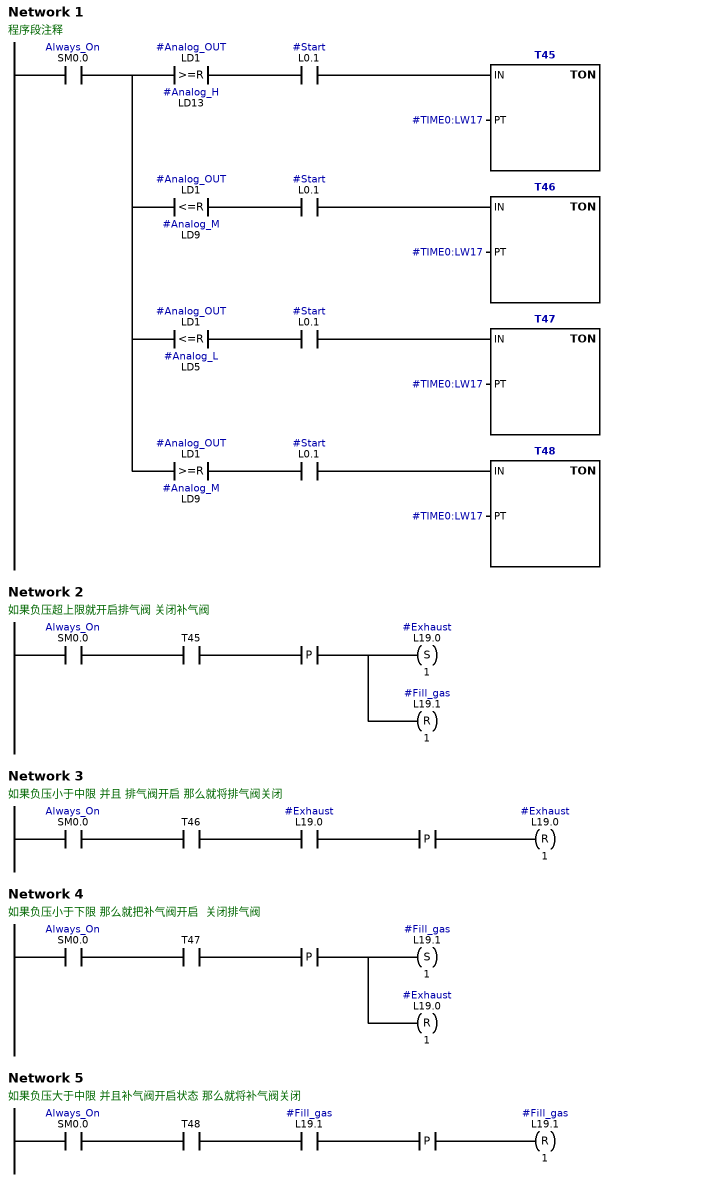
[picture p24: SBR13 networks 1-5]
Network 1
// 程序段注释
LD     Always_On:SM0.0
LPS
AR>=   #Analog_OUT:LD1, #Analog_H:LD13
A      #Start:L0.1
TON    T45, #TIME0:LW17
LRD
AR<=   #Analog_OUT:LD1, #Analog_M:LD9
A      #Start:L0.1
TON    T46, #TIME0:LW17
LRD
AR<=   #Analog_OUT:LD1, #Analog_L:LD5
A      #Start:L0.1
TON    T47, #TIME0:LW17
LPP
AR>=   #Analog_OUT:LD1, #Analog_M:LD9
A      #Start:L0.1
TON    T48, #TIME0:LW17
Network 2
// 如果负压超上限就开启排气阀 关闭补气阀
LD     Always_On:SM0.0
A      T45
EU
S      #Exhaust:L19.0, 1
R      #Fill_gas:L19.1, 1
Network 3
// 如果负压小于中限 并且 排气阀开启 那么就将排气阀关闭
LD     Always_On:SM0.0
A      T46
A      #Exhaust:L19.0
EU
R      #Exhaust:L19.0, 1
Network 4
// 如果负压小于下限 那么就把补气阀开启  关闭排气阀
LD     Always_On:SM0.0
A      T47
EU
S      #Fill_gas:L19.1, 1
R      #Exhaust:L19.0, 1
Network 5
// 如果负压大于中限 并且补气阀开启状态 那么就将补气阀关闭 
LD     Always_On:SM0.0
A      T48
A      #Fill_gas:L19.1
EU
R      #Fill_gas:L19.1, 1
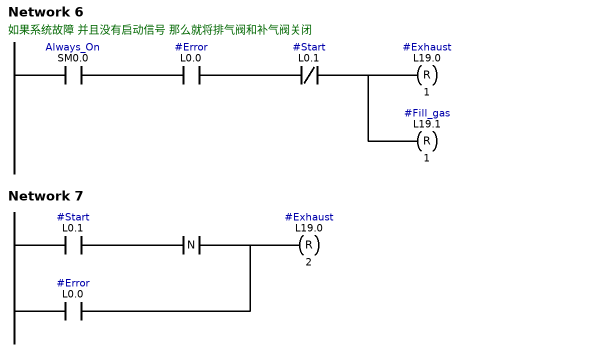
Network 6
// 如果系统故障 并且没有启动信号 那么就将排气阀和补气阀关闭
LD     Always_On:SM0.0
A      #Error:L0.0
AN     #Start:L0.1
R      #Exhaust:L19.0, 1
R      #Fill_gas:L19.1, 1
Network 7
LD     #Start:L0.1
ED
O      #Error:L0.0
R      #Exhaust:L19.0, 2
END_SUBROUTINE_BLOCK

SUBROUTINE_BLOCK 混料程序:SBR14
TITLE=1.	混合机启动程序:做按钮单独启停控制(实现批混模式)
// 
// 2.	混合机进料状态，达到重量大于1000kg（可调）延时ＸＸＳ
// 　　　    进入混合状态，停止输出混合要料信号．
// 
// 3.	混合状态（混合时间可调），显示混料时间，做倒计时。
// 
// 4.	混料完成信号，（运行出料）
// 
// 5.	出料达到设定出料下限下于100ｋｇ（可调）延时XXS，再次进入混料进料状态。
//                 需要显示混料机的状态，（进料，混合计时，出料）
// 
VAR_INPUT
Star:BOOL;	// L0.0 混合机启动
MixmotorWeight:DWORD;	// LD1 混合机重量读取
WeightH:DWORD;	// LD5 混合机重量上限
WeightL:DWORD;	// LD9 混合机重量下限
DelayH:WORD;	// LW13 上限延时
DelayL:WORD;	// LW15 下限延时
MixtimeSet:WORD;	// LW17 混合时间设置
END_VAR
VAR_IN_OUT
FeedState:BOOL;	// L19.0 进料状态
MixState:BOOL;	// L19.1 混合状态
OutState:BOOL;	// L19.2 出料状态
Countdown:WORD;	// LW20 混合倒计时
MixMotor:BOOL;	// L22.0 混合机电机
OutDone:BOOL;	// L22.1 出料完成
END_VAR
BEGIN
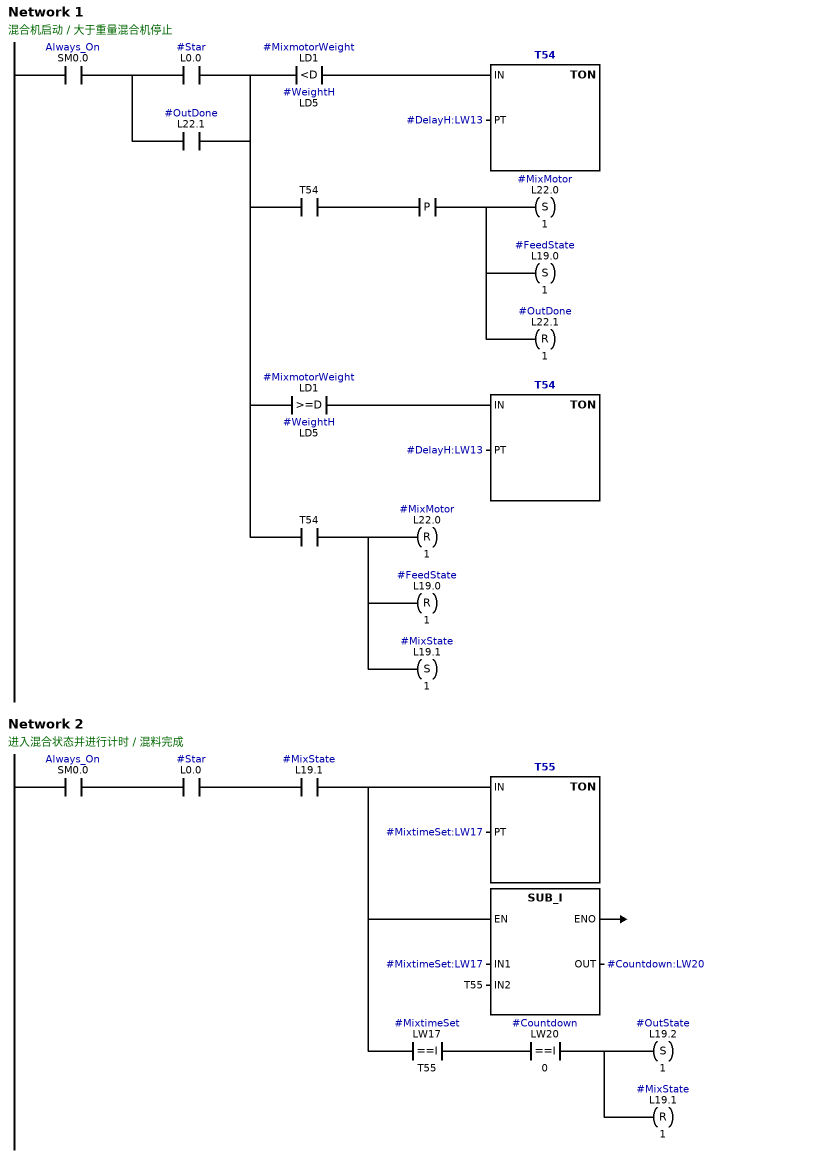
Network 1
// 混合机启动
// 大于重量混合机停止
LD     Always_On:SM0.0
LD     #Star:L0.0
O      #OutDone:L22.1
ALD
LPS
AD<    #MixmotorWeight:LD1, #WeightH:LD5
TON    T54, #DelayH:LW13
LRD
A      T54
EU
S      #MixMotor:L22.0, 1
S      #FeedState:L19.0, 1
R      #OutDone:L22.1, 1
LRD
AD>=   #MixmotorWeight:LD1, #WeightH:LD5
TON    T54, #DelayH:LW13
LPP
A      T54
R      #MixMotor:L22.0, 1
R      #FeedState:L19.0, 1
S      #MixState:L19.1, 1
Network 2
// 进入混合状态并进行计时
// 混料完成
LD     Always_On:SM0.0
A      #Star:L0.0
A      #MixState:L19.1
TON    T55, #MixtimeSet:LW17
MOVW   #MixtimeSet:LW17, #Countdown:LW20
-I     T55, #Countdown:LW20
AW=    #MixtimeSet:LW17, T55
AW=    #Countdown:LW20, 0
S      #OutState:L19.2, 1
R      #MixState:L19.1, 1
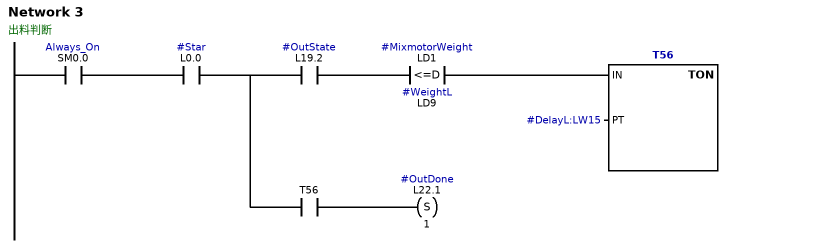
Network 3
// 出料判断
LD     Always_On:SM0.0
A      #Star:L0.0
LPS
A      #OutState:L19.2
AD<=   #MixmotorWeight:LD1, #WeightL:LD9
TON    T56, #DelayL:LW15
LPP
A      T56
S      #OutDone:L22.1, 1
END_SUBROUTINE_BLOCK

SUBROUTINE_BLOCK 系统泄压程序:SBR15
TITLE=
VAR_INPUT
Start:BOOL;	// L0.0 
OUT_Analog:REAL;	// LD1 
END_VAR
VAR_IN_OUT
Date_set_FH:REAL;	// LD5 
Date_set_FL:REAL;	// LD9 
Date_set_ZH:REAL;	// LD13 
Date_set_ZL:REAL;	// LD17 
Auto_OUT:BOOL;	// L21.0 
END_VAR
VAR
Auto_16A:BOOL;	// L21.1 中间变量1
Auto_16B:BOOL;	// L21.2 中间变量2
END_VAR
BEGIN
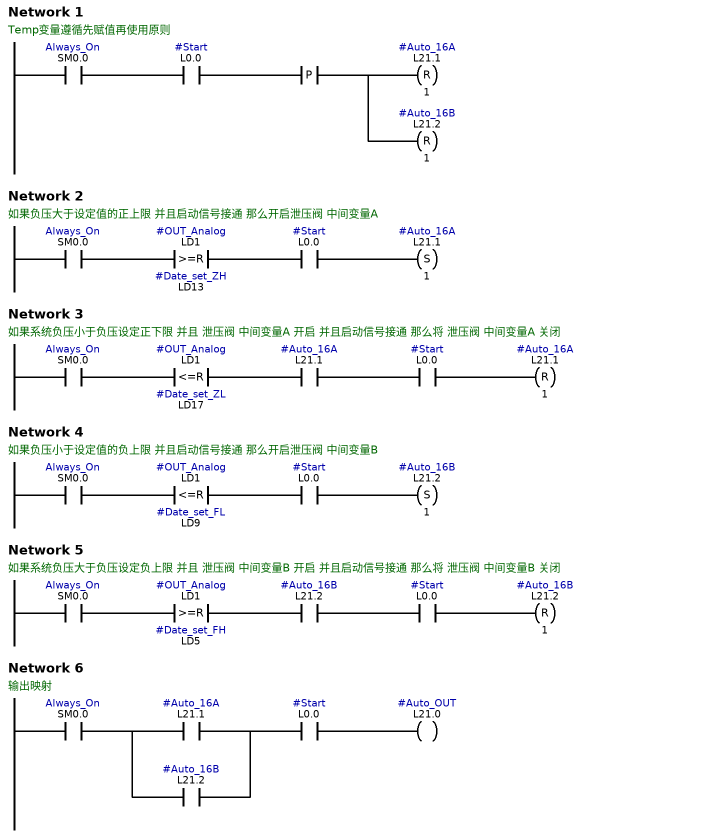
Network 1
// Temp变量遵循先赋值再使用原则
LD     Always_On:SM0.0
A      #Start:L0.0
EU
R      #Auto_16A:L21.1, 1
R      #Auto_16B:L21.2, 1
Network 2
// 如果负压大于设定值的正上限 并且启动信号接通 那么开启泄压阀 中间变量A
LD     Always_On:SM0.0
AR>=   #OUT_Analog:LD1, #Date_set_ZH:LD13
A      #Start:L0.0
S      #Auto_16A:L21.1, 1
Network 3
// 如果系统负压小于负压设定正下限 并且 泄压阀 中间变量A 开启 并且启动信号接通 那么将 泄压阀 中间变量A 关闭
LD     Always_On:SM0.0
AR<=   #OUT_Analog:LD1, #Date_set_ZL:LD17
A      #Auto_16A:L21.1
A      #Start:L0.0
R      #Auto_16A:L21.1, 1
Network 4
// 如果负压小于设定值的负上限 并且启动信号接通 那么开启泄压阀 中间变量B
LD     Always_On:SM0.0
AR<=   #OUT_Analog:LD1, #Date_set_FL:LD9
A      #Start:L0.0
S      #Auto_16B:L21.2, 1
Network 5
// 如果系统负压大于负压设定负上限 并且 泄压阀 中间变量B 开启 并且启动信号接通 那么将 泄压阀 中间变量B 关闭
LD     Always_On:SM0.0
AR>=   #OUT_Analog:LD1, #Date_set_FH:LD5
A      #Auto_16B:L21.2
A      #Start:L0.0
R      #Auto_16B:L21.2, 1
Network 6
// 输出映射
LD     Always_On:SM0.0
LD     #Auto_16A:L21.1
O      #Auto_16B:L21.2
ALD
A      #Start:L0.0
=      #Auto_OUT:L21.0
END_SUBROUTINE_BLOCK

SUBROUTINE_BLOCK 仓泵1:SBR16
TITLE=
VAR_INPUT
IN_LW:BOOL;	// L0.0 上料位信号
END_VAR
VAR_IN_OUT
呼吸阀:BOOL;	// L0.1 
进料阀:BOOL;	// L0.2 
进料阀上:BOOL;	// L0.3 
仓顶阀:BOOL;	// L0.4 
硫化阀:BOOL;	// L0.5 
输送阀:BOOL;	// L0.6 
疏通阀:BOOL;	// L0.7 
出口阀:BOOL;	// L1.0 
切换阀:BOOL;	// L1.1 
END_VAR
BEGIN
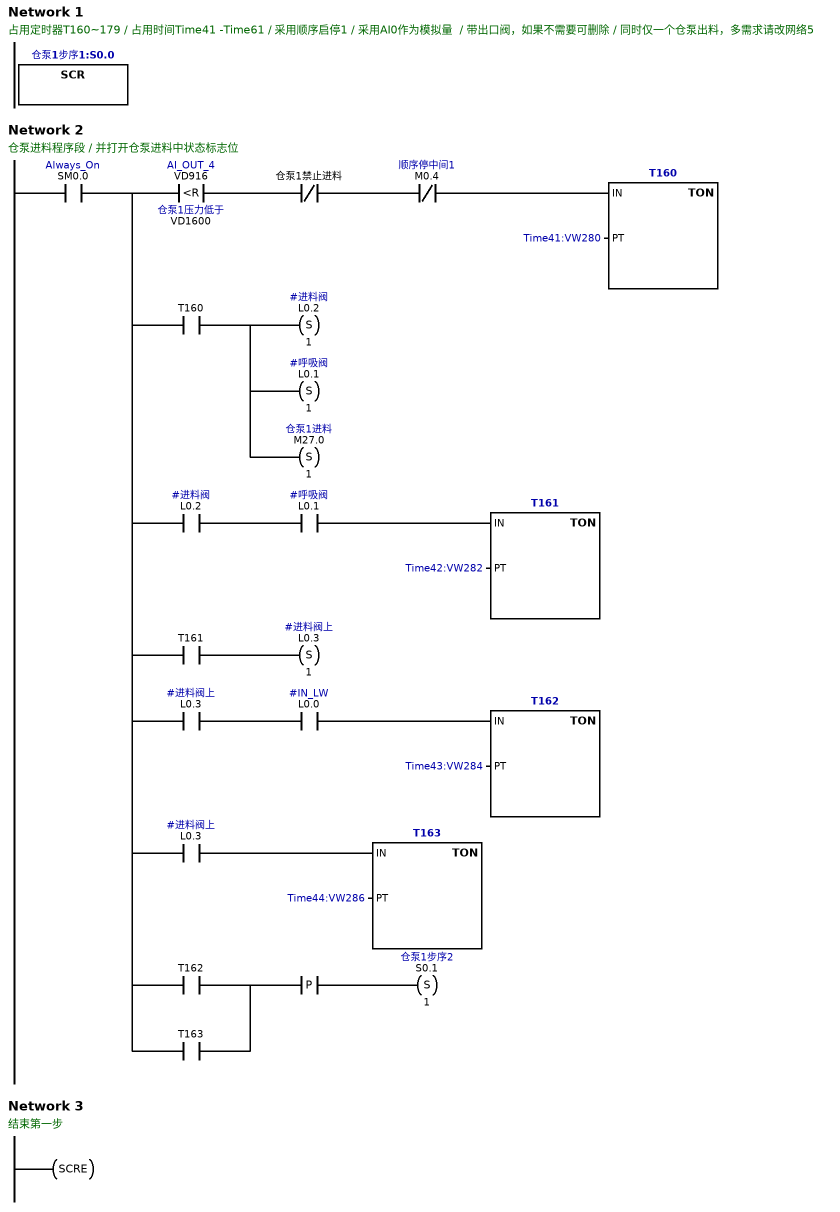
Network 1
// 占用定时器T160~179
// 占用时间Time41 -Time61
// 采用顺序启停1
// 采用AI0作为模拟量 
// 带出口阀，如果不需要可删除
// 同时仅一个仓泵出料，多需求请改网络5
LSCR   仓泵1步序1:S0.0
Network 2
// 仓泵进料程序段
// 并打开仓泵进料中状态标志位
// (network saved uncompiled; LAD cells follow)
// row 0: c0 -| |- Always_On:SM0.0 v  c1 -|<R|- AI_OUT_4:VD916, 仓泵1压力低于:VD1600  c2 -|/|- 仓泵1禁止进料  c3 -|/|- 顺序停中间1:M0.4  c4 --  c5 [TON T160 IN:=power@row0, PT:=Time41:VW280]
// row 1: c0 ^v  c5 [box]
// row 2: c0 ^v  c1 -| |- T160 v  c2 -(S) #进料阀:L0.2, 1
// row 3: c0 ^v  c1 ^v  c2 -(S) #呼吸阀:L0.1, 1
// row 4: c0 ^v  c1 ^  c2 -(S) 仓泵1进料:M27.0, 1
// row 5: c0 ^v  c1 -| |- #进料阀:L0.2  c2 -| |- #呼吸阀:L0.1  c3 --  c4 [TON T161 IN:=power@row5, PT:=Time42:VW282]
// row 6: c0 ^v  c4 [box]
// row 7: c0 ^v  c1 -| |- T161  c2 -(S) #进料阀上:L0.3, 1
// row 8: c0 ^v  c1 -| |- #进料阀上:L0.3  c2 -| |- #IN_LW:L0.0  c3 --  c4 [TON T162 IN:=power@row8, PT:=Time43:VW284]
// row 9: c0 ^v  c4 [box]
// row 10: c0 ^v  c1 -| |- #进料阀上:L0.3  c2 --  c3 [TON T163 IN:=power@row10, PT:=Time44:VW286]
// row 11: c0 ^v  c3 [box]
// row 12: c0 ^v  c1 -| |- T162 v  c2 -|P|-  c3 -(S) 仓泵1步序2:S0.1, 1
// row 13: c0 ^  c1 -| |- T163 ^
Network 3
// 结束第一步
SCRE
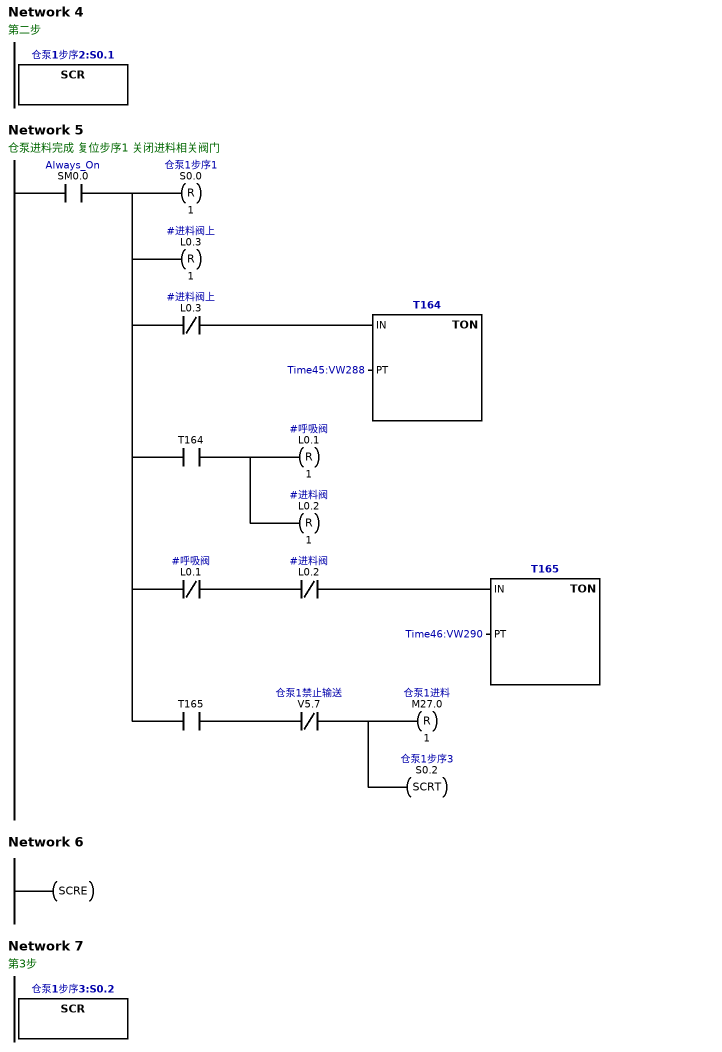
Network 4
// 第二步 
LSCR   仓泵1步序2:S0.1
Network 5
// 仓泵进料完成 复位步序1 关闭进料相关阀门
LD     Always_On:SM0.0
LPS
R      仓泵1步序1:S0.0, 1
R      #进料阀上:L0.3, 1
AN     #进料阀上:L0.3
TON    T164, Time45:VW288
LRD
A      T164
R      #呼吸阀:L0.1, 1
R      #进料阀:L0.2, 1
LRD
AN     #呼吸阀:L0.1
AN     #进料阀:L0.2
TON    T165, Time46:VW290
LPP
A      T165
AN     仓泵1禁止输送:V5.7
R      仓泵1进料:M27.0, 1
SCRT   仓泵1步序3:S0.2
Network 6
SCRE
Network 7
// 第3步 
LSCR   仓泵1步序3:S0.2
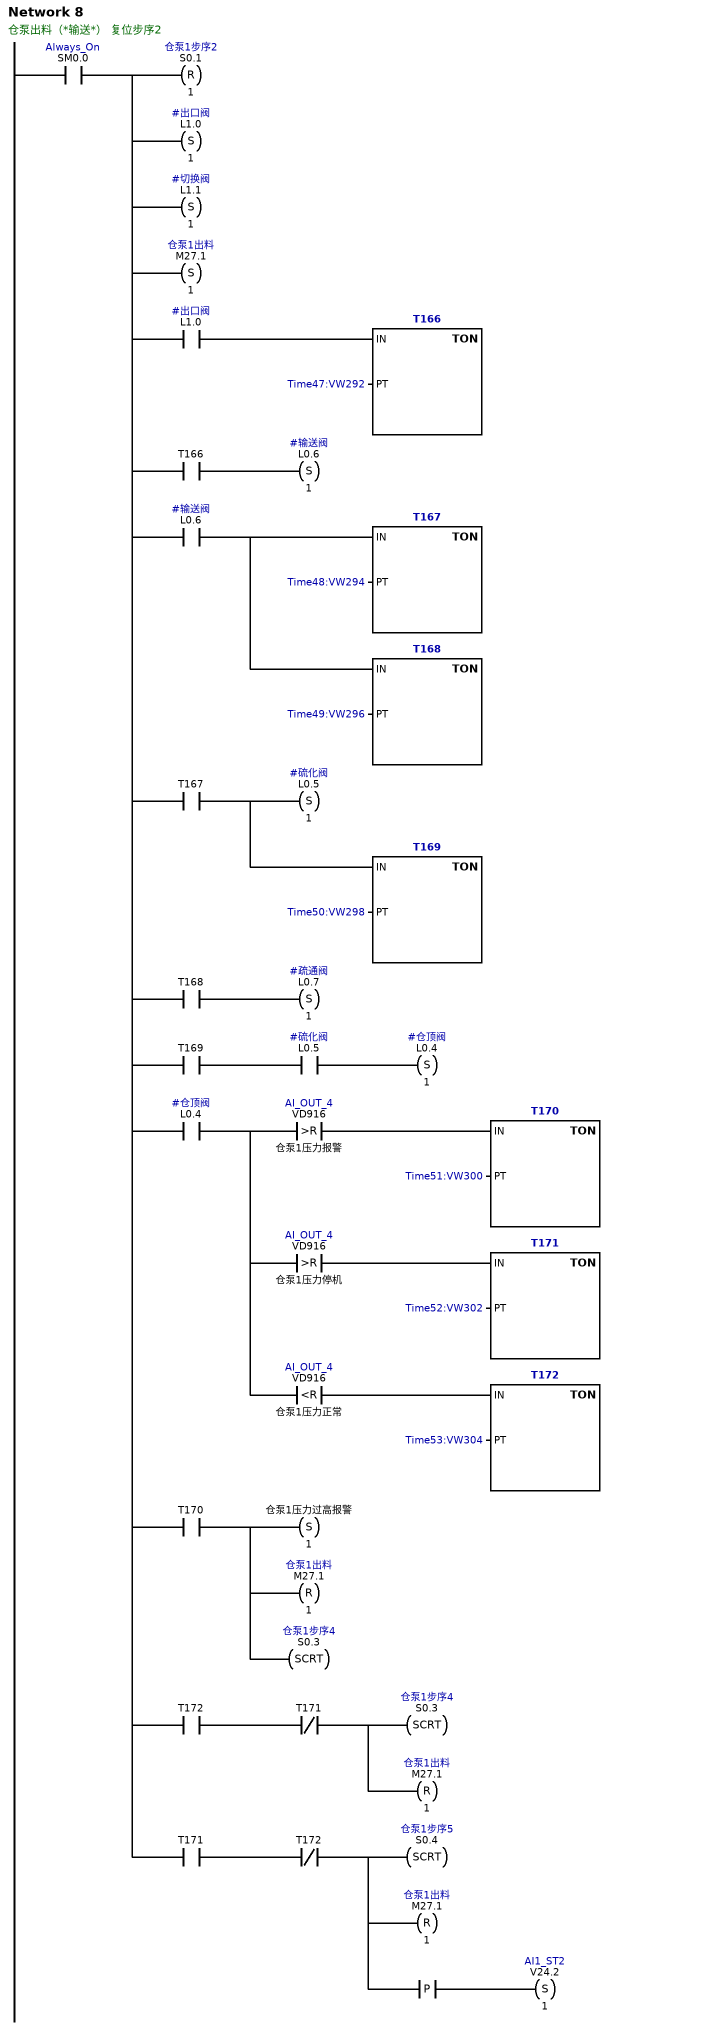
Network 8
// 仓泵出料（*输送*） 复位步序2
// (network saved uncompiled; LAD cells follow)
// row 0: c0 -| |- Always_On:SM0.0 v  c1 -(R) 仓泵1步序2:S0.1, 1
// row 1: c0 ^v  c1 -(S) #出口阀:L1.0, 1
// row 2: c0 ^v  c1 -(S) #切换阀:L1.1, 1
// row 3: c0 ^v  c1 -(S) 仓泵1出料:M27.1, 1
// row 4: c0 ^v  c1 -| |- #出口阀:L1.0  c2 --  c3 [TON T166 IN:=power@row4, PT:=Time47:VW292]
// row 5: c0 ^v  c3 [box]
// row 6: c0 ^v  c1 -| |- T166  c2 -(S) #输送阀:L0.6, 1
// row 7: c0 ^v  c1 -| |- #输送阀:L0.6 v  c2 --  c3 [TON T167 IN:=power@row7, PT:=Time48:VW294]
// row 8: c0 ^v  c1 ^v  c3 [box]
// row 9: c0 ^v  c1 ^  c2 --  c3 [TON T168 IN:=power@row9, PT:=Time49:VW296]
// row 10: c0 ^v  c3 [box]
// row 11: c0 ^v  c1 -| |- T167 v  c2 -(S) #硫化阀:L0.5, 1
// row 12: c0 ^v  c1 ^  c2 --  c3 [TON T169 IN:=power@row12, PT:=Time50:VW298]
// row 13: c0 ^v  c3 [box]
// row 14: c0 ^v  c1 -| |- T168  c2 -(S) #疏通阀:L0.7, 1
// row 15: c0 ^v  c1 -| |- T169  c2 -| |- #硫化阀:L0.5  c3 -(S) #仓顶阀:L0.4, 1
// row 16: c0 ^v  c1 -| |- #仓顶阀:L0.4 v  c2 -|>R|- AI_OUT_4:VD916, 仓泵1压力报警  c3 --  c4 [TON T170 IN:=power@row16, PT:=Time51:VW300]
// row 17: c0 ^v  c1 ^v  c4 [box]
// row 18: c0 ^v  c1 ^v  c2 -|>R|- AI_OUT_4:VD916, 仓泵1压力停机  c3 --  c4 [TON T171 IN:=power@row18, PT:=Time52:VW302]
// row 19: c0 ^v  c1 ^v  c4 [box]
// row 20: c0 ^v  c1 ^  c2 -|<R|- AI_OUT_4:VD916, 仓泵1压力正常  c3 --  c4 [TON T172 IN:=power@row20, PT:=Time53:VW304]
// row 21: c0 ^v  c4 [box]
// row 22: c0 ^v  c1 -| |- T170 v  c2 -(S) 仓泵1压力过高报警, 1
// row 23: c0 ^v  c1 ^v  c2 -(R) 仓泵1出料:M27.1, 1
// row 24: c0 ^v  c1 ^  c2 -(SCRT) 仓泵1步序4:S0.3
// row 25: c0 ^v  c1 -| |- T172  c2 -|/|- T171 v  c3 -(SCRT) 仓泵1步序4:S0.3
// row 26: c0 ^v  c2 ^  c3 -(R) 仓泵1出料:M27.1, 1
// row 27: c0 ^  c1 -| |- T171  c2 -|/|- T172 v  c3 -(SCRT) 仓泵1步序5:S0.4
// row 28: c2 ^v  c3 -(R) 仓泵1出料:M27.1, 1
// row 29: c2 ^  c3 -|P|-  c4 -(S) AI1_ST2:V24.2, 1
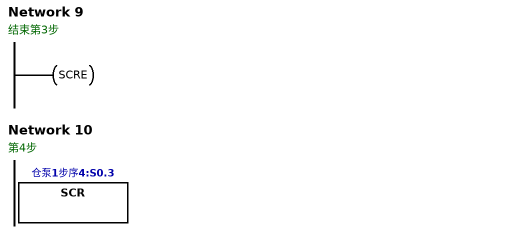
Network 9
// 结束第3步
SCRE
Network 10
// 第4步 
LSCR   仓泵1步序4:S0.3
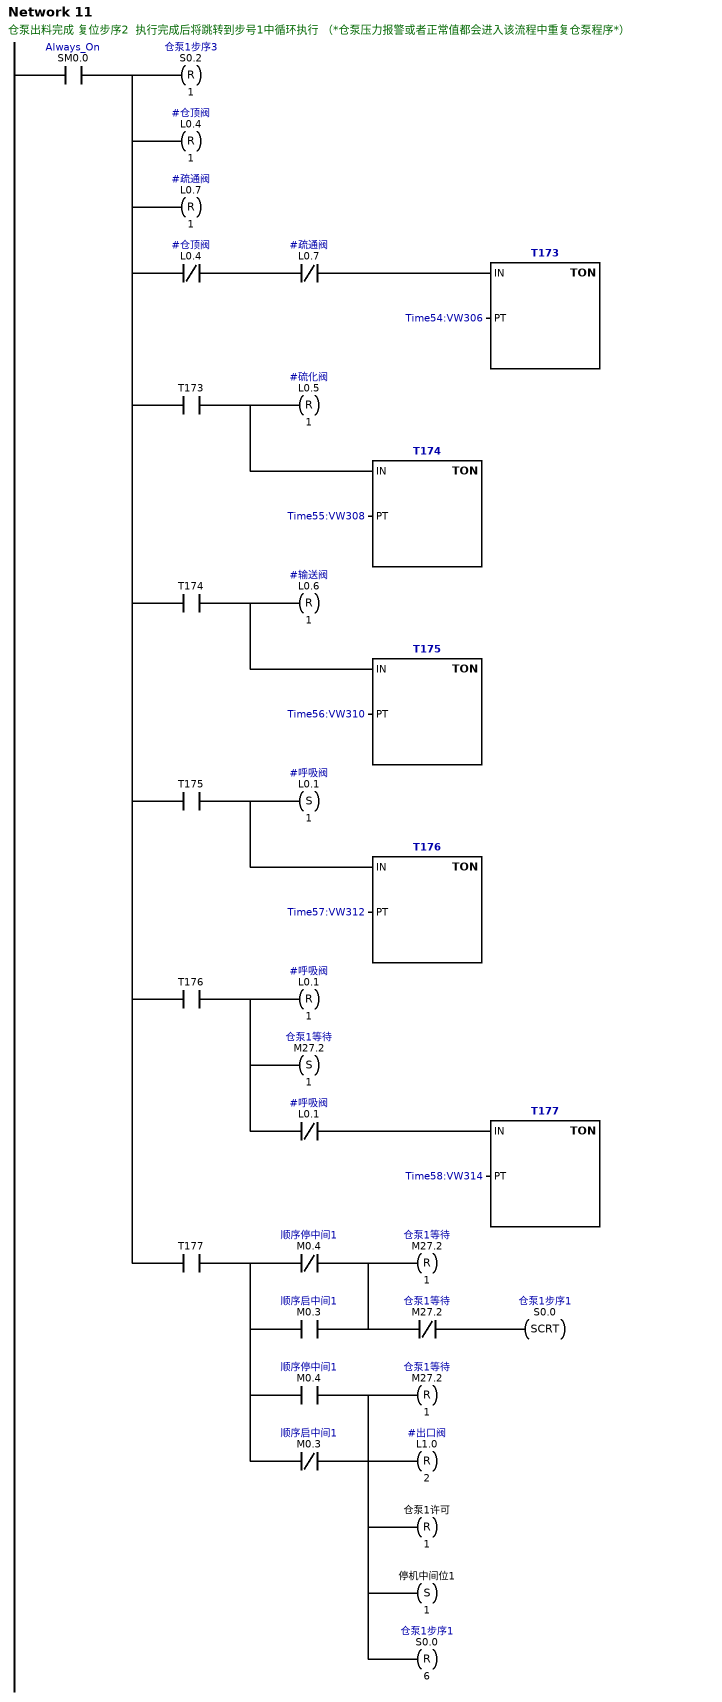
Network 11
// 仓泵出料完成 复位步序2  执行完成后将跳转到步号1中循环执行 （*仓泵压力报警或者正常值都会进入该流程中重复仓泵程序*）
// (network saved uncompiled; LAD cells follow)
// row 0: c0 -| |- Always_On:SM0.0 v  c1 -(R) 仓泵1步序3:S0.2, 1
// row 1: c0 ^v  c1 -(R) #仓顶阀:L0.4, 1
// row 2: c0 ^v  c1 -(R) #疏通阀:L0.7, 1
// row 3: c0 ^v  c1 -|/|- #仓顶阀:L0.4  c2 -|/|- #疏通阀:L0.7  c3 --  c4 [TON T173 IN:=power@row3, PT:=Time54:VW306]
// row 4: c0 ^v  c4 [box]
// row 5: c0 ^v  c1 -| |- T173 v  c2 -(R) #硫化阀:L0.5, 1
// row 6: c0 ^v  c1 ^  c2 --  c3 [TON T174 IN:=power@row6, PT:=Time55:VW308]
// row 7: c0 ^v  c3 [box]
// row 8: c0 ^v  c1 -| |- T174 v  c2 -(R) #输送阀:L0.6, 1
// row 9: c0 ^v  c1 ^  c2 --  c3 [TON T175 IN:=power@row9, PT:=Time56:VW310]
// row 10: c0 ^v  c3 [box]
// row 11: c0 ^v  c1 -| |- T175 v  c2 -(S) #呼吸阀:L0.1, 1
// row 12: c0 ^v  c1 ^  c2 --  c3 [TON T176 IN:=power@row12, PT:=Time57:VW312]
// row 13: c0 ^v  c3 [box]
// row 14: c0 ^v  c1 -| |- T176 v  c2 -(R) #呼吸阀:L0.1, 1
// row 15: c0 ^v  c1 ^v  c2 -(S) 仓泵1等待:M27.2, 1
// row 16: c0 ^v  c1 ^  c2 -|/|- #呼吸阀:L0.1  c3 --  c4 [TON T177 IN:=power@row16, PT:=Time58:VW314]
// row 17: c0 ^v  c4 [box]
// row 18: c0 ^  c1 -| |- T177 v  c2 -|/|- 顺序停中间1:M0.4 v  c3 -(R) 仓泵1等待:M27.2, 1
// row 19: c1 ^v  c2 -| |- 顺序启中间1:M0.3 ^  c3 -|/|- 仓泵1等待:M27.2  c4 -(SCRT) 仓泵1步序1:S0.0
// row 20: c1 ^v  c2 -| |- 顺序停中间1:M0.4 v  c3 -(R) 仓泵1等待:M27.2, 1
// row 21: c1 ^  c2 -|/|- 顺序启中间1:M0.3 ^v  c3 -(R) #出口阀:L1.0, 2
// row 22: c2 ^v  c3 -(R) 仓泵1许可, 1
// row 23: c2 ^v  c3 -(S) 停机中间位1, 1
// row 24: c2 ^  c3 -(R) 仓泵1步序1:S0.0, 6
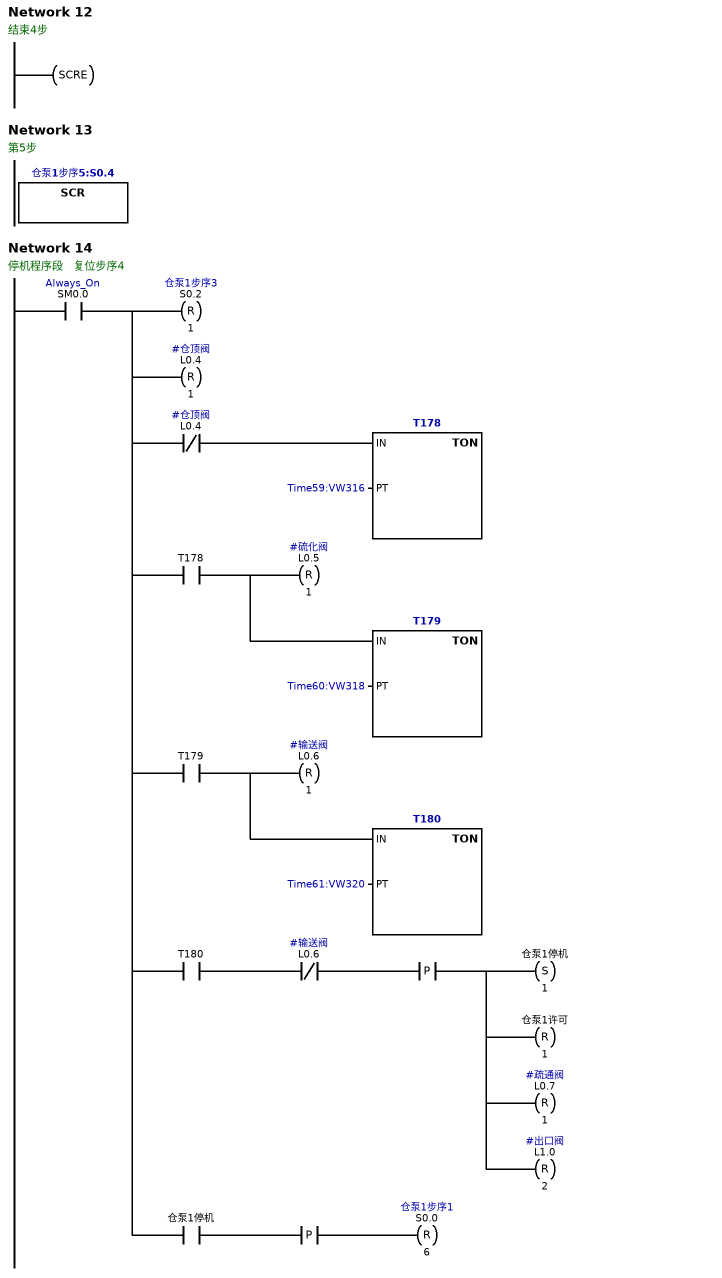
Network 12
// 结束4步
SCRE
Network 13
// 第5步 
LSCR   仓泵1步序5:S0.4
Network 14
// 停机程序段   复位步序4 
// (network saved uncompiled; LAD cells follow)
// row 0: c0 -| |- Always_On:SM0.0 v  c1 -(R) 仓泵1步序3:S0.2, 1
// row 1: c0 ^v  c1 -(R) #仓顶阀:L0.4, 1
// row 2: c0 ^v  c1 -|/|- #仓顶阀:L0.4  c2 --  c3 [TON T178 IN:=power@row2, PT:=Time59:VW316]
// row 3: c0 ^v  c3 [box]
// row 4: c0 ^v  c1 -| |- T178 v  c2 -(R) #硫化阀:L0.5, 1
// row 5: c0 ^v  c1 ^  c2 --  c3 [TON T179 IN:=power@row5, PT:=Time60:VW318]
// row 6: c0 ^v  c3 [box]
// row 7: c0 ^v  c1 -| |- T179 v  c2 -(R) #输送阀:L0.6, 1
// row 8: c0 ^v  c1 ^  c2 --  c3 [TON T180 IN:=power@row8, PT:=Time61:VW320]
// row 9: c0 ^v  c3 [box]
// row 10: c0 ^v  c1 -| |- T180  c2 -|/|- #输送阀:L0.6  c3 -|P|-  v  c4 -(S) 仓泵1停机, 1
// row 11: c0 ^v  c3 ^v  c4 -(R) 仓泵1许可, 1
// row 12: c0 ^v  c3 ^v  c4 -(R) #疏通阀:L0.7, 1
// row 13: c0 ^v  c3 ^  c4 -(R) #出口阀:L1.0, 2
// row 14: c0 ^  c1 -| |- 仓泵1停机  c2 -|P|-  c3 -(R) 仓泵1步序1:S0.0, 6
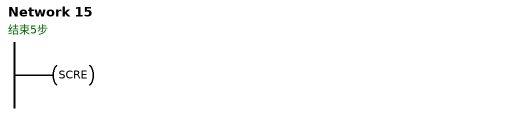
Network 15
// 结束5步
SCRE
END_SUBROUTINE_BLOCK

SUBROUTINE_BLOCK 仓泵2:SBR17
TITLE=
VAR_INPUT
IN_LW:BOOL;	// L0.0 上料位信号
END_VAR
VAR_IN_OUT
呼吸阀:BOOL;	// L0.1 
进料阀:BOOL;	// L0.2 
进料阀上:BOOL;	// L0.3 
仓顶阀:BOOL;	// L0.4 
硫化阀:BOOL;	// L0.5 
输送阀:BOOL;	// L0.6 
疏通阀:BOOL;	// L0.7 
出口阀:BOOL;	// L1.0 
切换阀:BOOL;	// L1.1 
END_VAR
BEGIN
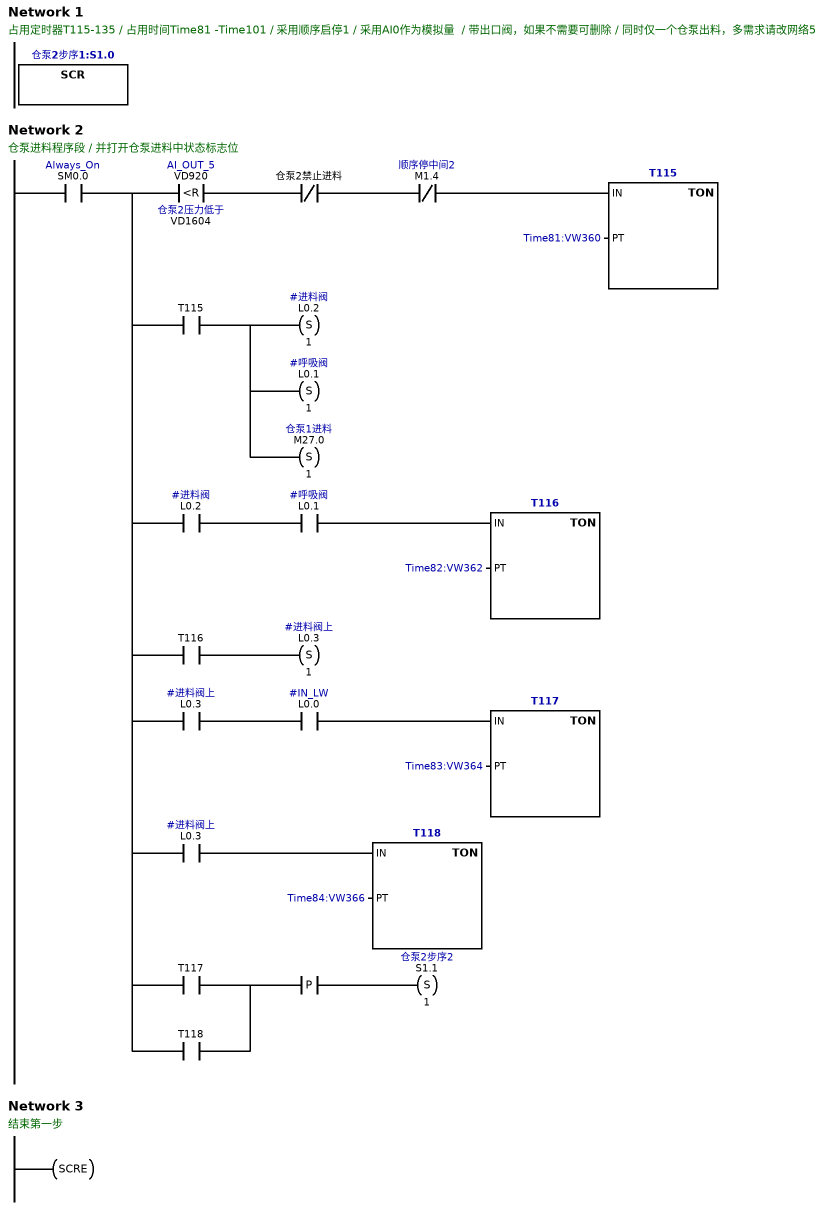
Network 1
// 占用定时器T115-135
// 占用时间Time81 -Time101
// 采用顺序启停1
// 采用AI0作为模拟量 
// 带出口阀，如果不需要可删除
// 同时仅一个仓泵出料，多需求请改网络5
LSCR   仓泵2步序1:S1.0
Network 2
// 仓泵进料程序段
// 并打开仓泵进料中状态标志位
// (network saved uncompiled; LAD cells follow)
// row 0: c0 -| |- Always_On:SM0.0 v  c1 -|<R|- AI_OUT_5:VD920, 仓泵2压力低于:VD1604  c2 -|/|- 仓泵2禁止进料  c3 -|/|- 顺序停中间2:M1.4  c4 --  c5 [TON T115 IN:=power@row0, PT:=Time81:VW360]
// row 1: c0 ^v  c5 [box]
// row 2: c0 ^v  c1 -| |- T115 v  c2 -(S) #进料阀:L0.2, 1
// row 3: c0 ^v  c1 ^v  c2 -(S) #呼吸阀:L0.1, 1
// row 4: c0 ^v  c1 ^  c2 -(S) 仓泵1进料:M27.0, 1
// row 5: c0 ^v  c1 -| |- #进料阀:L0.2  c2 -| |- #呼吸阀:L0.1  c3 --  c4 [TON T116 IN:=power@row5, PT:=Time82:VW362]
// row 6: c0 ^v  c4 [box]
// row 7: c0 ^v  c1 -| |- T116  c2 -(S) #进料阀上:L0.3, 1
// row 8: c0 ^v  c1 -| |- #进料阀上:L0.3  c2 -| |- #IN_LW:L0.0  c3 --  c4 [TON T117 IN:=power@row8, PT:=Time83:VW364]
// row 9: c0 ^v  c4 [box]
// row 10: c0 ^v  c1 -| |- #进料阀上:L0.3  c2 --  c3 [TON T118 IN:=power@row10, PT:=Time84:VW366]
// row 11: c0 ^v  c3 [box]
// row 12: c0 ^v  c1 -| |- T117 v  c2 -|P|-  c3 -(S) 仓泵2步序2:S1.1, 1
// row 13: c0 ^  c1 -| |- T118 ^
Network 3
// 结束第一步
SCRE
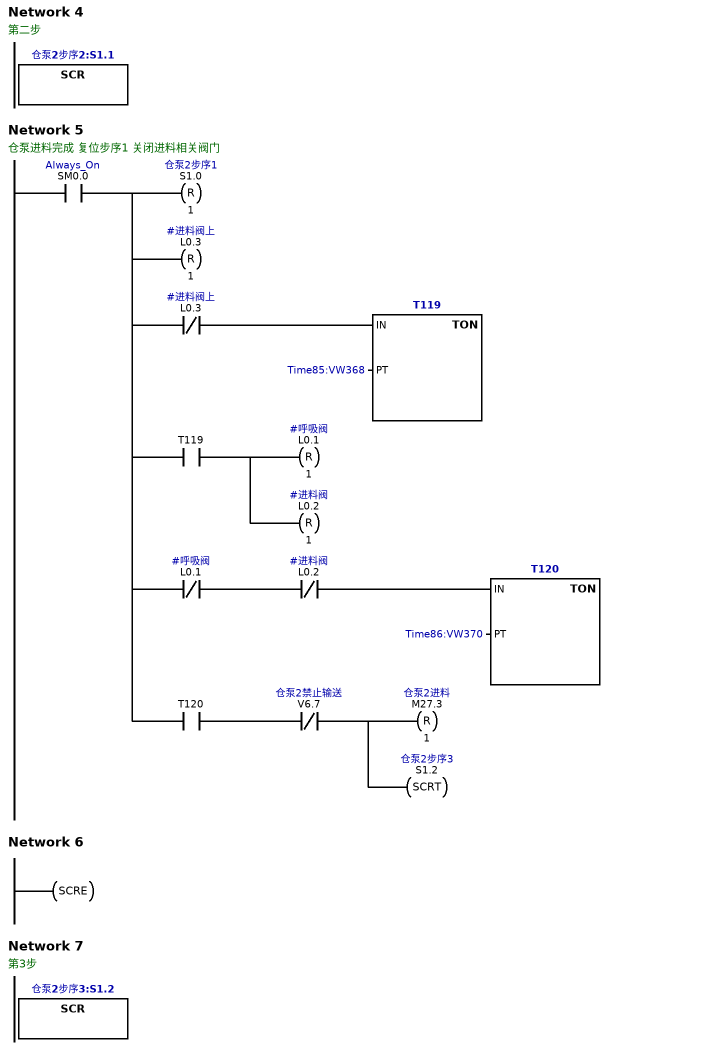
Network 4
// 第二步 
LSCR   仓泵2步序2:S1.1
Network 5
// 仓泵进料完成 复位步序1 关闭进料相关阀门
LD     Always_On:SM0.0
LPS
R      仓泵2步序1:S1.0, 1
R      #进料阀上:L0.3, 1
AN     #进料阀上:L0.3
TON    T119, Time85:VW368
LRD
A      T119
R      #呼吸阀:L0.1, 1
R      #进料阀:L0.2, 1
LRD
AN     #呼吸阀:L0.1
AN     #进料阀:L0.2
TON    T120, Time86:VW370
LPP
A      T120
AN     仓泵2禁止输送:V6.7
R      仓泵2进料:M27.3, 1
SCRT   仓泵2步序3:S1.2
Network 6
SCRE
Network 7
// 第3步 
LSCR   仓泵2步序3:S1.2
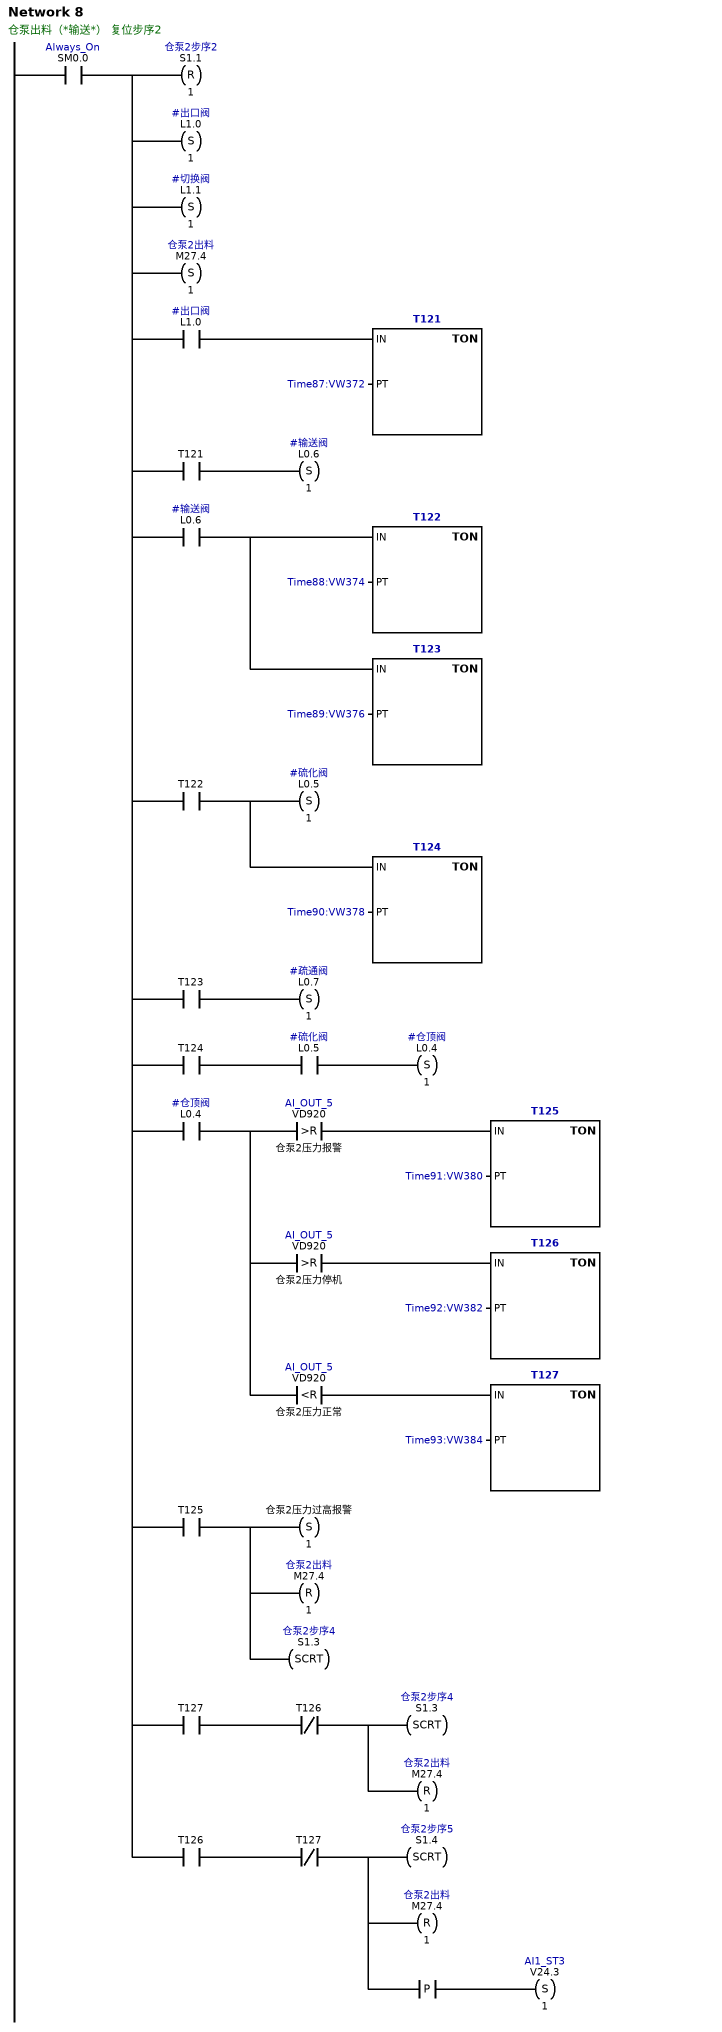
Network 8
// 仓泵出料（*输送*） 复位步序2
// (network saved uncompiled; LAD cells follow)
// row 0: c0 -| |- Always_On:SM0.0 v  c1 -(R) 仓泵2步序2:S1.1, 1
// row 1: c0 ^v  c1 -(S) #出口阀:L1.0, 1
// row 2: c0 ^v  c1 -(S) #切换阀:L1.1, 1
// row 3: c0 ^v  c1 -(S) 仓泵2出料:M27.4, 1
// row 4: c0 ^v  c1 -| |- #出口阀:L1.0  c2 --  c3 [TON T121 IN:=power@row4, PT:=Time87:VW372]
// row 5: c0 ^v  c3 [box]
// row 6: c0 ^v  c1 -| |- T121  c2 -(S) #输送阀:L0.6, 1
// row 7: c0 ^v  c1 -| |- #输送阀:L0.6 v  c2 --  c3 [TON T122 IN:=power@row7, PT:=Time88:VW374]
// row 8: c0 ^v  c1 ^v  c3 [box]
// row 9: c0 ^v  c1 ^  c2 --  c3 [TON T123 IN:=power@row9, PT:=Time89:VW376]
// row 10: c0 ^v  c3 [box]
// row 11: c0 ^v  c1 -| |- T122 v  c2 -(S) #硫化阀:L0.5, 1
// row 12: c0 ^v  c1 ^  c2 --  c3 [TON T124 IN:=power@row12, PT:=Time90:VW378]
// row 13: c0 ^v  c3 [box]
// row 14: c0 ^v  c1 -| |- T123  c2 -(S) #疏通阀:L0.7, 1
// row 15: c0 ^v  c1 -| |- T124  c2 -| |- #硫化阀:L0.5  c3 -(S) #仓顶阀:L0.4, 1
// row 16: c0 ^v  c1 -| |- #仓顶阀:L0.4 v  c2 -|>R|- AI_OUT_5:VD920, 仓泵2压力报警  c3 --  c4 [TON T125 IN:=power@row16, PT:=Time91:VW380]
// row 17: c0 ^v  c1 ^v  c4 [box]
// row 18: c0 ^v  c1 ^v  c2 -|>R|- AI_OUT_5:VD920, 仓泵2压力停机  c3 --  c4 [TON T126 IN:=power@row18, PT:=Time92:VW382]
// row 19: c0 ^v  c1 ^v  c4 [box]
// row 20: c0 ^v  c1 ^  c2 -|<R|- AI_OUT_5:VD920, 仓泵2压力正常  c3 --  c4 [TON T127 IN:=power@row20, PT:=Time93:VW384]
// row 21: c0 ^v  c4 [box]
// row 22: c0 ^v  c1 -| |- T125 v  c2 -(S) 仓泵2压力过高报警, 1
// row 23: c0 ^v  c1 ^v  c2 -(R) 仓泵2出料:M27.4, 1
// row 24: c0 ^v  c1 ^  c2 -(SCRT) 仓泵2步序4:S1.3
// row 25: c0 ^v  c1 -| |- T127  c2 -|/|- T126 v  c3 -(SCRT) 仓泵2步序4:S1.3
// row 26: c0 ^v  c2 ^  c3 -(R) 仓泵2出料:M27.4, 1
// row 27: c0 ^  c1 -| |- T126  c2 -|/|- T127 v  c3 -(SCRT) 仓泵2步序5:S1.4
// row 28: c2 ^v  c3 -(R) 仓泵2出料:M27.4, 1
// row 29: c2 ^  c3 -|P|-  c4 -(S) AI1_ST3:V24.3, 1
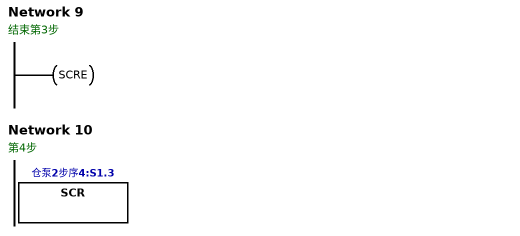
Network 9
// 结束第3步
SCRE
Network 10
// 第4步 
LSCR   仓泵2步序4:S1.3
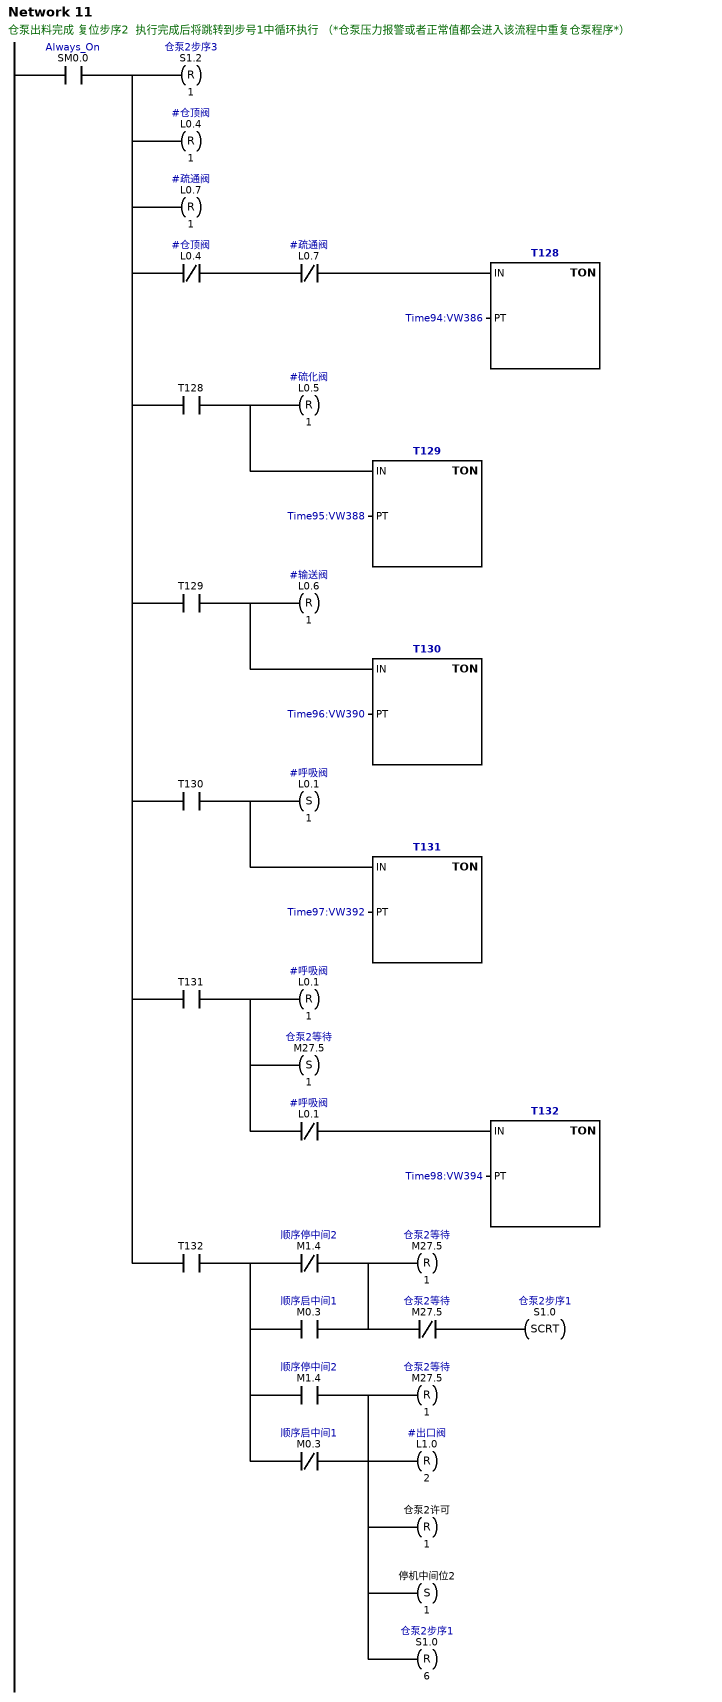
Network 11
// 仓泵出料完成 复位步序2  执行完成后将跳转到步号1中循环执行 （*仓泵压力报警或者正常值都会进入该流程中重复仓泵程序*）
// (network saved uncompiled; LAD cells follow)
// row 0: c0 -| |- Always_On:SM0.0 v  c1 -(R) 仓泵2步序3:S1.2, 1
// row 1: c0 ^v  c1 -(R) #仓顶阀:L0.4, 1
// row 2: c0 ^v  c1 -(R) #疏通阀:L0.7, 1
// row 3: c0 ^v  c1 -|/|- #仓顶阀:L0.4  c2 -|/|- #疏通阀:L0.7  c3 --  c4 [TON T128 IN:=power@row3, PT:=Time94:VW386]
// row 4: c0 ^v  c4 [box]
// row 5: c0 ^v  c1 -| |- T128 v  c2 -(R) #硫化阀:L0.5, 1
// row 6: c0 ^v  c1 ^  c2 --  c3 [TON T129 IN:=power@row6, PT:=Time95:VW388]
// row 7: c0 ^v  c3 [box]
// row 8: c0 ^v  c1 -| |- T129 v  c2 -(R) #输送阀:L0.6, 1
// row 9: c0 ^v  c1 ^  c2 --  c3 [TON T130 IN:=power@row9, PT:=Time96:VW390]
// row 10: c0 ^v  c3 [box]
// row 11: c0 ^v  c1 -| |- T130 v  c2 -(S) #呼吸阀:L0.1, 1
// row 12: c0 ^v  c1 ^  c2 --  c3 [TON T131 IN:=power@row12, PT:=Time97:VW392]
// row 13: c0 ^v  c3 [box]
// row 14: c0 ^v  c1 -| |- T131 v  c2 -(R) #呼吸阀:L0.1, 1
// row 15: c0 ^v  c1 ^v  c2 -(S) 仓泵2等待:M27.5, 1
// row 16: c0 ^v  c1 ^  c2 -|/|- #呼吸阀:L0.1  c3 --  c4 [TON T132 IN:=power@row16, PT:=Time98:VW394]
// row 17: c0 ^v  c4 [box]
// row 18: c0 ^  c1 -| |- T132 v  c2 -|/|- 顺序停中间2:M1.4 v  c3 -(R) 仓泵2等待:M27.5, 1
// row 19: c1 ^v  c2 -| |- 顺序启中间1:M0.3 ^  c3 -|/|- 仓泵2等待:M27.5  c4 -(SCRT) 仓泵2步序1:S1.0
// row 20: c1 ^v  c2 -| |- 顺序停中间2:M1.4 v  c3 -(R) 仓泵2等待:M27.5, 1
// row 21: c1 ^  c2 -|/|- 顺序启中间1:M0.3 ^v  c3 -(R) #出口阀:L1.0, 2
// row 22: c2 ^v  c3 -(R) 仓泵2许可, 1
// row 23: c2 ^v  c3 -(S) 停机中间位2, 1
// row 24: c2 ^  c3 -(R) 仓泵2步序1:S1.0, 6
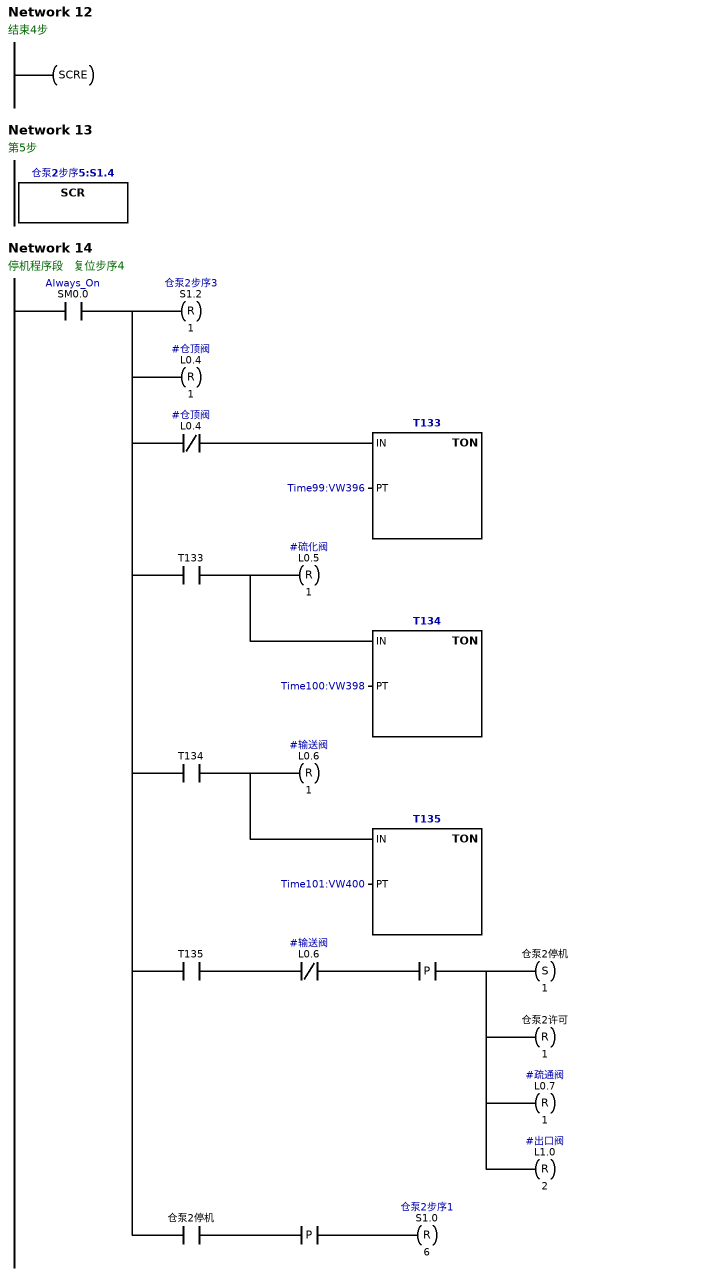
Network 12
// 结束4步
SCRE
Network 13
// 第5步 
LSCR   仓泵2步序5:S1.4
Network 14
// 停机程序段   复位步序4 
// (network saved uncompiled; LAD cells follow)
// row 0: c0 -| |- Always_On:SM0.0 v  c1 -(R) 仓泵2步序3:S1.2, 1
// row 1: c0 ^v  c1 -(R) #仓顶阀:L0.4, 1
// row 2: c0 ^v  c1 -|/|- #仓顶阀:L0.4  c2 --  c3 [TON T133 IN:=power@row2, PT:=Time99:VW396]
// row 3: c0 ^v  c3 [box]
// row 4: c0 ^v  c1 -| |- T133 v  c2 -(R) #硫化阀:L0.5, 1
// row 5: c0 ^v  c1 ^  c2 --  c3 [TON T134 IN:=power@row5, PT:=Time100:VW398]
// row 6: c0 ^v  c3 [box]
// row 7: c0 ^v  c1 -| |- T134 v  c2 -(R) #输送阀:L0.6, 1
// row 8: c0 ^v  c1 ^  c2 --  c3 [TON T135 IN:=power@row8, PT:=Time101:VW400]
// row 9: c0 ^v  c3 [box]
// row 10: c0 ^v  c1 -| |- T135  c2 -|/|- #输送阀:L0.6  c3 -|P|-  v  c4 -(S) 仓泵2停机, 1
// row 11: c0 ^v  c3 ^v  c4 -(R) 仓泵2许可, 1
// row 12: c0 ^v  c3 ^v  c4 -(R) #疏通阀:L0.7, 1
// row 13: c0 ^v  c3 ^  c4 -(R) #出口阀:L1.0, 2
// row 14: c0 ^  c1 -| |- 仓泵2停机  c2 -|P|-  c3 -(R) 仓泵2步序1:S1.0, 6
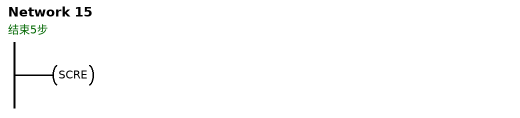
Network 15
// 结束5步
SCRE
END_SUBROUTINE_BLOCK

SUBROUTINE_BLOCK 仓泵3:SBR18
TITLE=
VAR_INPUT
IN_LW:BOOL;	// L0.0 上料位信号
END_VAR
VAR_IN_OUT
出口阀1:BOOL;	// L0.1 
出口阀2:BOOL;	// L0.2 
呼吸阀:BOOL;	// L0.3 
进料阀:BOOL;	// L0.4 
进料阀上:BOOL;	// L0.5 
仓顶阀:BOOL;	// L0.6 
硫化阀:BOOL;	// L0.7 
输送阀:BOOL;	// L1.0 
疏通阀:BOOL;	// L1.1 
END_VAR
BEGIN
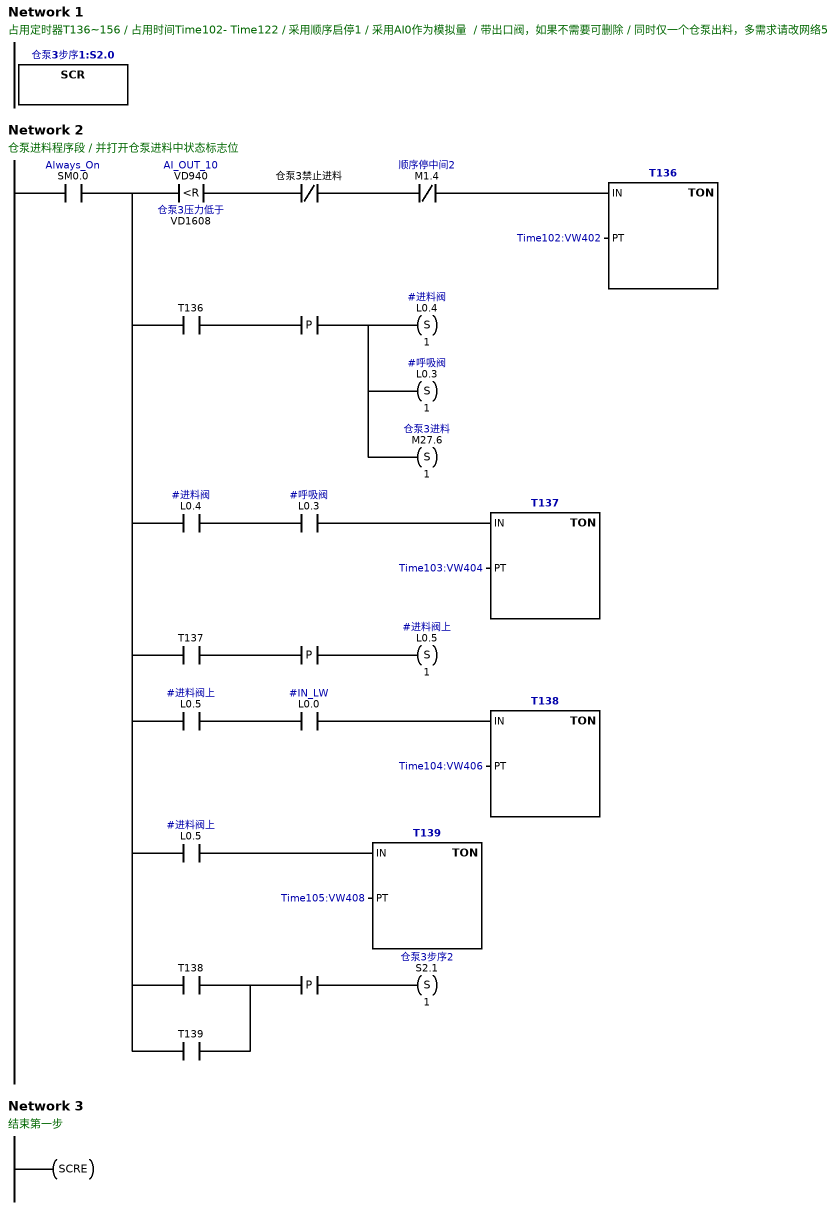
Network 1
// 占用定时器T136~156
// 占用时间Time102- Time122
// 采用顺序启停1
// 采用AI0作为模拟量 
// 带出口阀，如果不需要可删除
// 同时仅一个仓泵出料，多需求请改网络5
LSCR   仓泵3步序1:S2.0
Network 2
// 仓泵进料程序段
// 并打开仓泵进料中状态标志位
// (network saved uncompiled; LAD cells follow)
// row 0: c0 -| |- Always_On:SM0.0 v  c1 -|<R|- AI_OUT_10:VD940, 仓泵3压力低于:VD1608  c2 -|/|- 仓泵3禁止进料  c3 -|/|- 顺序停中间2:M1.4  c4 --  c5 [TON T136 IN:=power@row0, PT:=Time102:VW402]
// row 1: c0 ^v  c5 [box]
// row 2: c0 ^v  c1 -| |- T136  c2 -|P|-  v  c3 -(S) #进料阀:L0.4, 1
// row 3: c0 ^v  c2 ^v  c3 -(S) #呼吸阀:L0.3, 1
// row 4: c0 ^v  c2 ^  c3 -(S) 仓泵3进料:M27.6, 1
// row 5: c0 ^v  c1 -| |- #进料阀:L0.4  c2 -| |- #呼吸阀:L0.3  c3 --  c4 [TON T137 IN:=power@row5, PT:=Time103:VW404]
// row 6: c0 ^v  c4 [box]
// row 7: c0 ^v  c1 -| |- T137  c2 -|P|-  c3 -(S) #进料阀上:L0.5, 1
// row 8: c0 ^v  c1 -| |- #进料阀上:L0.5  c2 -| |- #IN_LW:L0.0  c3 --  c4 [TON T138 IN:=power@row8, PT:=Time104:VW406]
// row 9: c0 ^v  c4 [box]
// row 10: c0 ^v  c1 -| |- #进料阀上:L0.5  c2 --  c3 [TON T139 IN:=power@row10, PT:=Time105:VW408]
// row 11: c0 ^v  c3 [box]
// row 12: c0 ^v  c1 -| |- T138 v  c2 -|P|-  c3 -(S) 仓泵3步序2:S2.1, 1
// row 13: c0 ^  c1 -| |- T139 ^
Network 3
// 结束第一步
SCRE
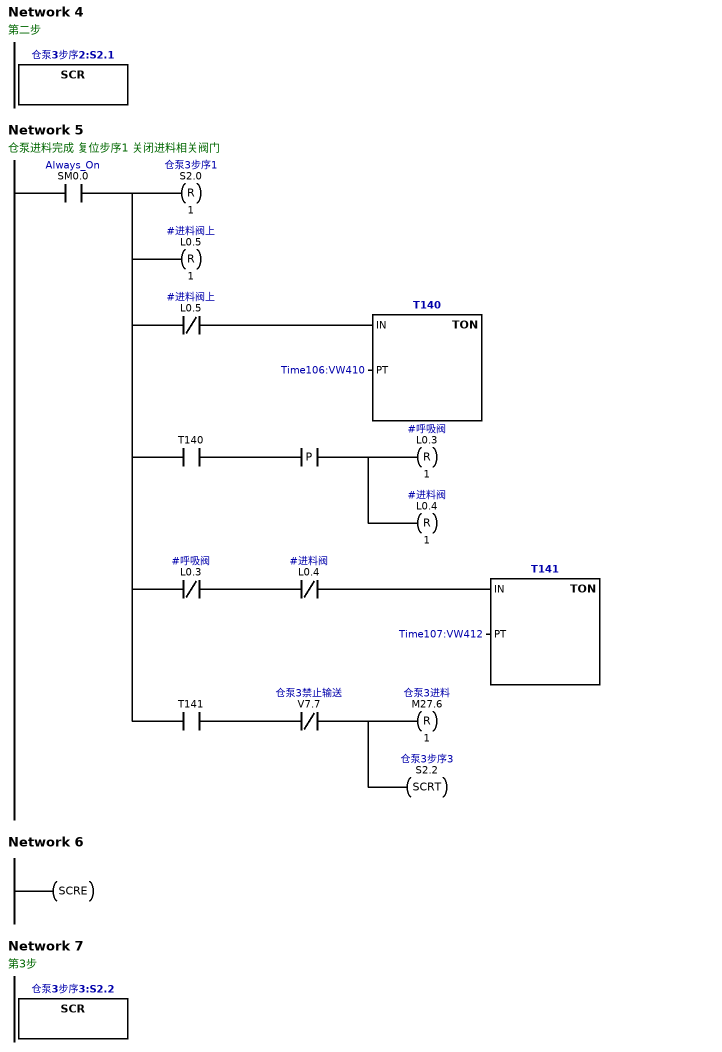
Network 4
// 第二步 
LSCR   仓泵3步序2:S2.1
Network 5
// 仓泵进料完成 复位步序1 关闭进料相关阀门
LD     Always_On:SM0.0
LPS
R      仓泵3步序1:S2.0, 1
R      #进料阀上:L0.5, 1
AN     #进料阀上:L0.5
TON    T140, Time106:VW410
LRD
A      T140
EU
R      #呼吸阀:L0.3, 1
R      #进料阀:L0.4, 1
LRD
AN     #呼吸阀:L0.3
AN     #进料阀:L0.4
TON    T141, Time107:VW412
LPP
A      T141
AN     仓泵3禁止输送:V7.7
R      仓泵3进料:M27.6, 1
SCRT   仓泵3步序3:S2.2
Network 6
SCRE
Network 7
// 第3步 
LSCR   仓泵3步序3:S2.2
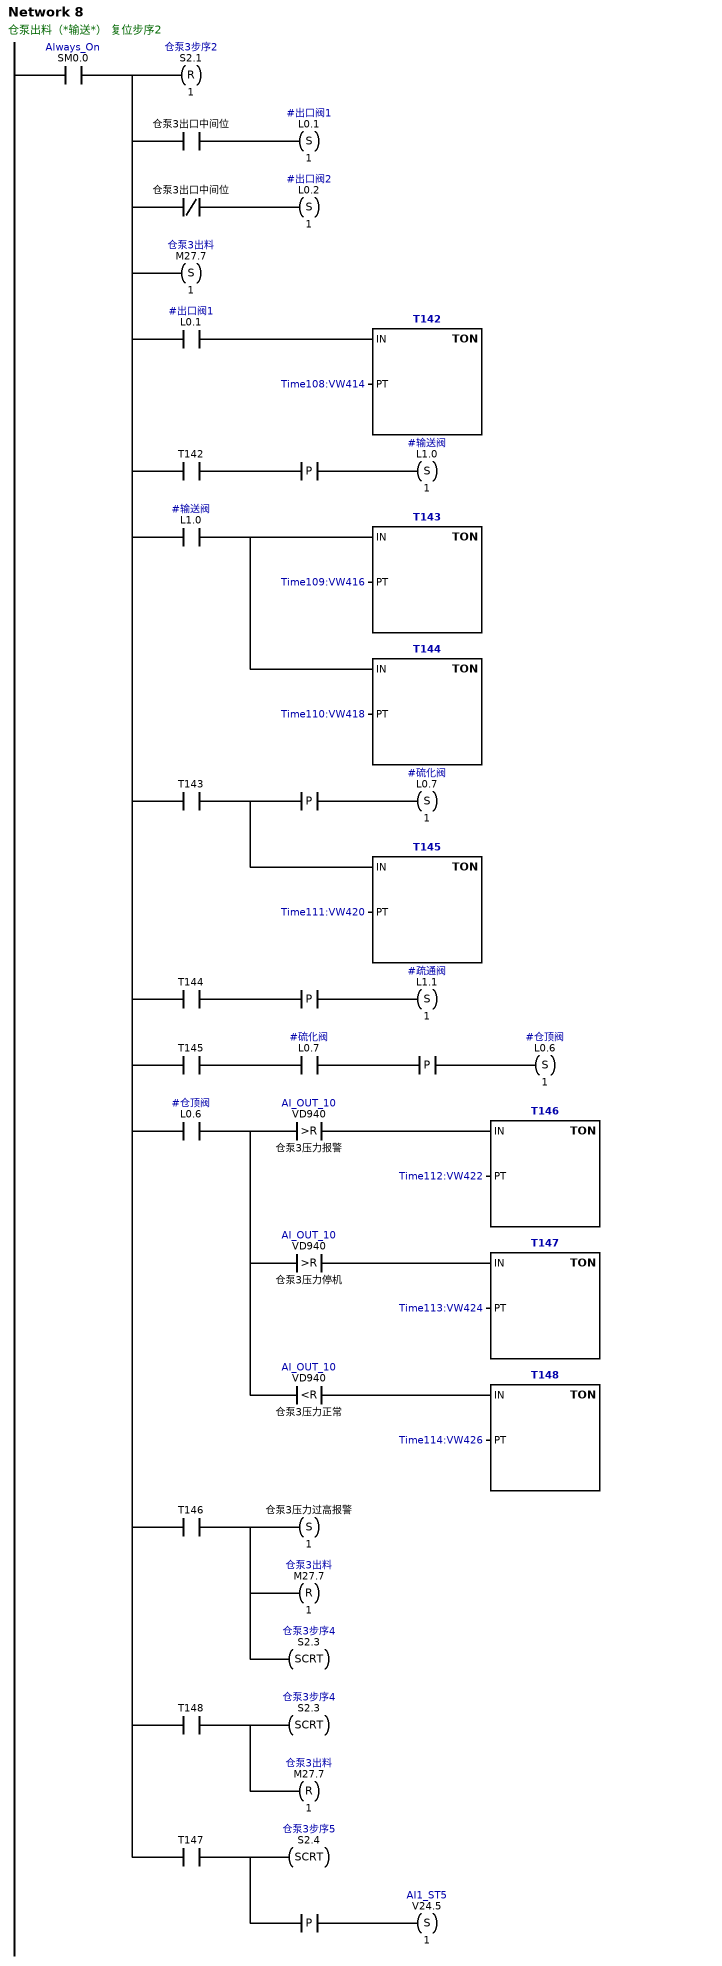
Network 8
// 仓泵出料（*输送*） 复位步序2
// (network saved uncompiled; LAD cells follow)
// row 0: c0 -| |- Always_On:SM0.0 v  c1 -(R) 仓泵3步序2:S2.1, 1
// row 1: c0 ^v  c1 -| |- 仓泵3出口中间位  c2 -(S) #出口阀1:L0.1, 1
// row 2: c0 ^v  c1 -|/|- 仓泵3出口中间位  c2 -(S) #出口阀2:L0.2, 1
// row 3: c0 ^v  c1 -(S) 仓泵3出料:M27.7, 1
// row 4: c0 ^v  c1 -| |- #出口阀1:L0.1  c2 --  c3 [TON T142 IN:=power@row4, PT:=Time108:VW414]
// row 5: c0 ^v  c3 [box]
// row 6: c0 ^v  c1 -| |- T142  c2 -|P|-  c3 -(S) #输送阀:L1.0, 1
// row 7: c0 ^v  c1 -| |- #输送阀:L1.0 v  c2 --  c3 [TON T143 IN:=power@row7, PT:=Time109:VW416]
// row 8: c0 ^v  c1 ^v  c3 [box]
// row 9: c0 ^v  c1 ^  c2 --  c3 [TON T144 IN:=power@row9, PT:=Time110:VW418]
// row 10: c0 ^v  c3 [box]
// row 11: c0 ^v  c1 -| |- T143 v  c2 -|P|-  c3 -(S) #硫化阀:L0.7, 1
// row 12: c0 ^v  c1 ^  c2 --  c3 [TON T145 IN:=power@row12, PT:=Time111:VW420]
// row 13: c0 ^v  c3 [box]
// row 14: c0 ^v  c1 -| |- T144  c2 -|P|-  c3 -(S) #疏通阀:L1.1, 1
// row 15: c0 ^v  c1 -| |- T145  c2 -| |- #硫化阀:L0.7  c3 -|P|-  c4 -(S) #仓顶阀:L0.6, 1
// row 16: c0 ^v  c1 -| |- #仓顶阀:L0.6 v  c2 -|>R|- AI_OUT_10:VD940, 仓泵3压力报警  c3 --  c4 [TON T146 IN:=power@row16, PT:=Time112:VW422]
// row 17: c0 ^v  c1 ^v  c4 [box]
// row 18: c0 ^v  c1 ^v  c2 -|>R|- AI_OUT_10:VD940, 仓泵3压力停机  c3 --  c4 [TON T147 IN:=power@row18, PT:=Time113:VW424]
// row 19: c0 ^v  c1 ^v  c4 [box]
// row 20: c0 ^v  c1 ^  c2 -|<R|- AI_OUT_10:VD940, 仓泵3压力正常  c3 --  c4 [TON T148 IN:=power@row20, PT:=Time114:VW426]
// row 21: c0 ^v  c4 [box]
// row 22: c0 ^v  c1 -| |- T146 v  c2 -(S) 仓泵3压力过高报警, 1
// row 23: c0 ^v  c1 ^v  c2 -(R) 仓泵3出料:M27.7, 1
// row 24: c0 ^v  c1 ^  c2 -(SCRT) 仓泵3步序4:S2.3
// row 25: c0 ^v  c1 -| |- T148 v  c2 -(SCRT) 仓泵3步序4:S2.3
// row 26: c0 ^v  c1 ^  c2 -(R) 仓泵3出料:M27.7, 1
// row 27: c0 ^  c1 -| |- T147 v  c2 -(SCRT) 仓泵3步序5:S2.4
// row 28: c1 ^  c2 -|P|-  c3 -(S) AI1_ST5:V24.5, 1
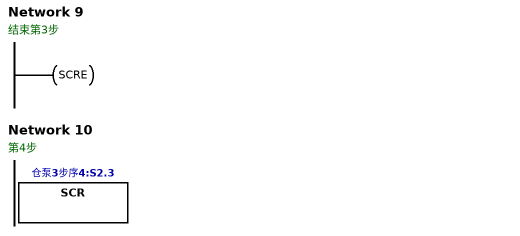
Network 9
// 结束第3步
SCRE
Network 10
// 第4步 
LSCR   仓泵3步序4:S2.3
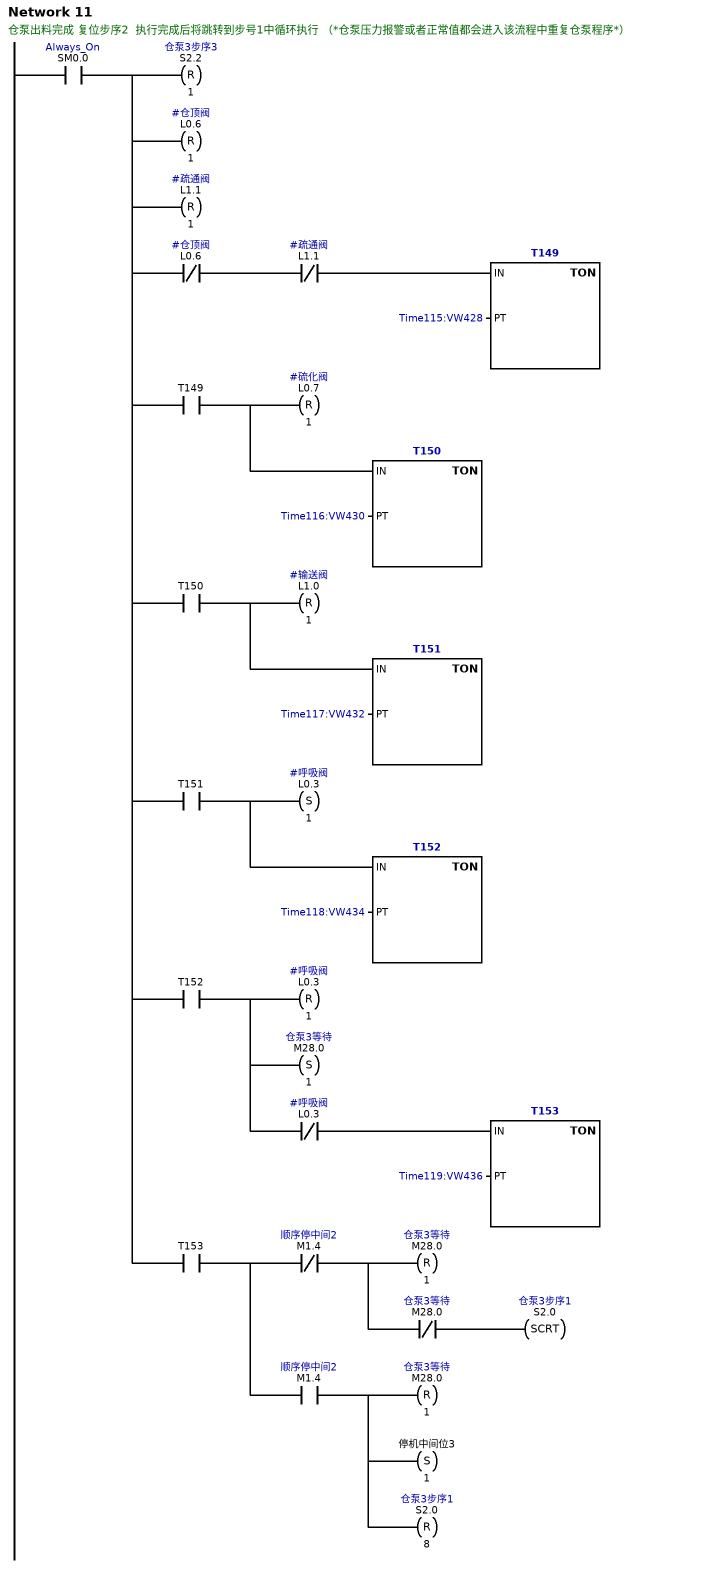
Network 11
// 仓泵出料完成 复位步序2  执行完成后将跳转到步号1中循环执行 （*仓泵压力报警或者正常值都会进入该流程中重复仓泵程序*）
// (network saved uncompiled; LAD cells follow)
// row 0: c0 -| |- Always_On:SM0.0 v  c1 -(R) 仓泵3步序3:S2.2, 1
// row 1: c0 ^v  c1 -(R) #仓顶阀:L0.6, 1
// row 2: c0 ^v  c1 -(R) #疏通阀:L1.1, 1
// row 3: c0 ^v  c1 -|/|- #仓顶阀:L0.6  c2 -|/|- #疏通阀:L1.1  c3 --  c4 [TON T149 IN:=power@row3, PT:=Time115:VW428]
// row 4: c0 ^v  c4 [box]
// row 5: c0 ^v  c1 -| |- T149 v  c2 -(R) #硫化阀:L0.7, 1
// row 6: c0 ^v  c1 ^  c2 --  c3 [TON T150 IN:=power@row6, PT:=Time116:VW430]
// row 7: c0 ^v  c3 [box]
// row 8: c0 ^v  c1 -| |- T150 v  c2 -(R) #输送阀:L1.0, 1
// row 9: c0 ^v  c1 ^  c2 --  c3 [TON T151 IN:=power@row9, PT:=Time117:VW432]
// row 10: c0 ^v  c3 [box]
// row 11: c0 ^v  c1 -| |- T151 v  c2 -(S) #呼吸阀:L0.3, 1
// row 12: c0 ^v  c1 ^  c2 --  c3 [TON T152 IN:=power@row12, PT:=Time118:VW434]
// row 13: c0 ^v  c3 [box]
// row 14: c0 ^v  c1 -| |- T152 v  c2 -(R) #呼吸阀:L0.3, 1
// row 15: c0 ^v  c1 ^v  c2 -(S) 仓泵3等待:M28.0, 1
// row 16: c0 ^v  c1 ^  c2 -|/|- #呼吸阀:L0.3  c3 --  c4 [TON T153 IN:=power@row16, PT:=Time119:VW436]
// row 17: c0 ^v  c4 [box]
// row 18: c0 ^  c1 -| |- T153 v  c2 -|/|- 顺序停中间2:M1.4 v  c3 -(R) 仓泵3等待:M28.0, 1
// row 19: c1 ^v  c2 ^  c3 -|/|- 仓泵3等待:M28.0  c4 -(SCRT) 仓泵3步序1:S2.0
// row 20: c1 ^  c2 -| |- 顺序停中间2:M1.4 v  c3 -(R) 仓泵3等待:M28.0, 1
// row 21: c2 ^v  c3 -(S) 停机中间位3, 1
// row 22: c2 ^  c3 -(R) 仓泵3步序1:S2.0, 8
